{attribute 'GeneratedUsingTerminal: EK1100-0000-0018'}
{attribute addProperty BoxType "EK1100-0000-0018"}
{attribute addProperty Id "Beckhoff_EJ4xxxEK1122Beckhoff_EJ4xxxEK1122_E11BF0B62A_0001_EJ4002_0000_0017EJ4002_18EC9E6515A_0002_EJ4002_0000_0018EJ4002_5AE37D9115A_0003_EJ4004_0000_0020EJ4004_D2A7C9B719A_0004_EJ4008_0000_0020EJ4008_01F55E9D27A_0005_EJ4018_0000_0016EJ4018_01F55E9D27A_0006_EJ4024_0000_0020EJ4024_D2A7C9B719A_0007_EJ4132_0000_0019EJ4132_18EC9E6515A_0008_EJ4134_0000_0019EJ4134_15C7AA1419A_0009_EJ4134_0000_0020EJ4134_15C7AA1419"}
{attribute addProperty CRC "2705704571"}
{attribute addProperty Size "177"}
TYPE Beckhoff_EJ4xxx_A145C67B EXTENDS EK1100_1FC0878B :
STRUCT
	{attribute addProperty Name "Beckhoff_EJ4xxxEK1122"}
	Beckhoff_EJ4xxxEK1122 : Beckhoff_EJ4xxxEK1122_E11BF0B6;
	{attribute addProperty Name "A_0001_EJ4002_0000_0017"}
	A_0001_EJ4002_0000_0017 : EJ4002_18EC9E65;
	{attribute addProperty Name "A_0002_EJ4002_0000_0018"}
	A_0002_EJ4002_0000_0018 : EJ4002_5AE37D91;
	{attribute addProperty Name "A_0003_EJ4004_0000_0020"}
	A_0003_EJ4004_0000_0020 : EJ4004_D2A7C9B7;
	{attribute addProperty Name "A_0004_EJ4008_0000_0020"}
	A_0004_EJ4008_0000_0020 : EJ4008_01F55E9D;
	{attribute addProperty Name "A_0005_EJ4018_0000_0016"}
	A_0005_EJ4018_0000_0016 : EJ4018_01F55E9D;
	{attribute addProperty Name "A_0006_EJ4024_0000_0020"}
	A_0006_EJ4024_0000_0020 : EJ4024_D2A7C9B7;
	{attribute addProperty Name "A_0007_EJ4132_0000_0019"}
	A_0007_EJ4132_0000_0019 : EJ4132_18EC9E65;
	{attribute addProperty Name "A_0008_EJ4134_0000_0019"}
	A_0008_EJ4134_0000_0019 : EJ4134_15C7AA14;
	{attribute addProperty Name "A_0009_EJ4134_0000_0020"}
	A_0009_EJ4134_0000_0020 : EJ4134_15C7AA14;
END_STRUCT
END_TYPE

(* stored: Version 1.2.0.0, ProductVersion 3.1.4024.9
   DUT Beckhoff_EJ4xxx_A145C67B: Id {45c3d464-a264-4637-af1f-461015f04683} *)
